FUNCTION_BLOCK cfb_controller
  (* Standard: 61499-2 *)
  (* Version 0.1, 2018-00-07, hpea485, UOA *)
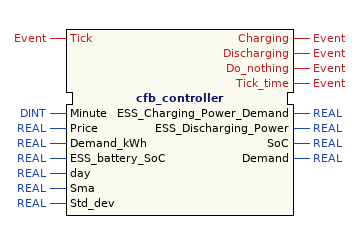
  EVENT_INPUT
    Tick;
  END_EVENT
  EVENT_OUTPUT
    Charging;
    Discharging;
    Do_nothing;
    Tick_time;
  END_EVENT
  VAR_INPUT
    Minute : DINT;
    Price : REAL;
    Demand_kWh : REAL;
    ESS_battery_SoC : REAL;
    day : REAL;
    Sma : REAL;
    Std_dev : REAL;
  END_VAR
  VAR_OUTPUT
    ESS_Charging_Power_Demand : REAL;
    ESS_Discharging_Power : REAL;
    SoC : REAL;
    Demand : REAL;
  END_VAR
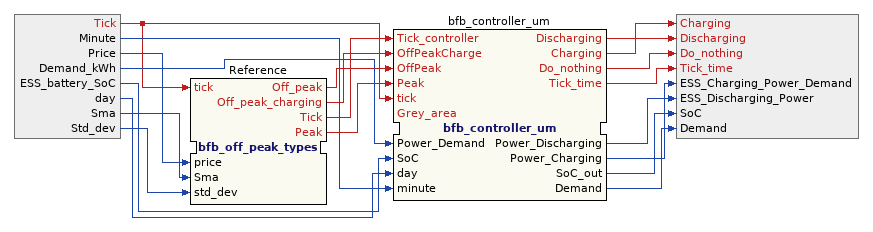
  FBS
    bfb_controller_um : bfb_controller_um;
    Reference : bfb_off_peak_types;
  END_FBS
  EVENT_CONNECTIONS
    Tick TO bfb_controller_um.tick;
    Tick TO Reference.tick;
    bfb_controller_um.Charging TO Charging;
    bfb_controller_um.Discharging TO Discharging;
    bfb_controller_um.Do_nothing TO Do_nothing;
    bfb_controller_um.Tick_time TO Tick_time;
    Reference.Off_peak TO bfb_controller_um.OffPeak;
    Reference.Off_peak_charging TO bfb_controller_um.OffPeakCharge;
    Reference.Tick TO bfb_controller_um.Tick_controller;
    Reference.Peak TO bfb_controller_um.Peak;
  END_CONNECTIONS
  DATA_CONNECTIONS
    Minute TO bfb_controller_um.minute;
    Price TO Reference.price;
    Demand_kWh TO bfb_controller_um.Power_Demand;
    ESS_battery_SoC TO bfb_controller_um.SoC;
    day TO bfb_controller_um.day;
    Sma TO Reference.Sma;
    Std_dev TO Reference.std_dev;
    bfb_controller_um.Power_Charging TO ESS_Charging_Power_Demand;
    bfb_controller_um.Power_Discharging TO ESS_Discharging_Power;
    bfb_controller_um.SoC_out TO SoC;
    bfb_controller_um.Demand TO Demand;
  END_CONNECTIONS
END_FUNCTION_BLOCK
